Staubli VAL3: start.pgx

program start()
begin
  call RobotMotion()
end
